SYSTEM TestMixerMain
  (* Version 1.0, 2024-03-03, ADMIN *)
  APPLICATION TestMixerMainApp
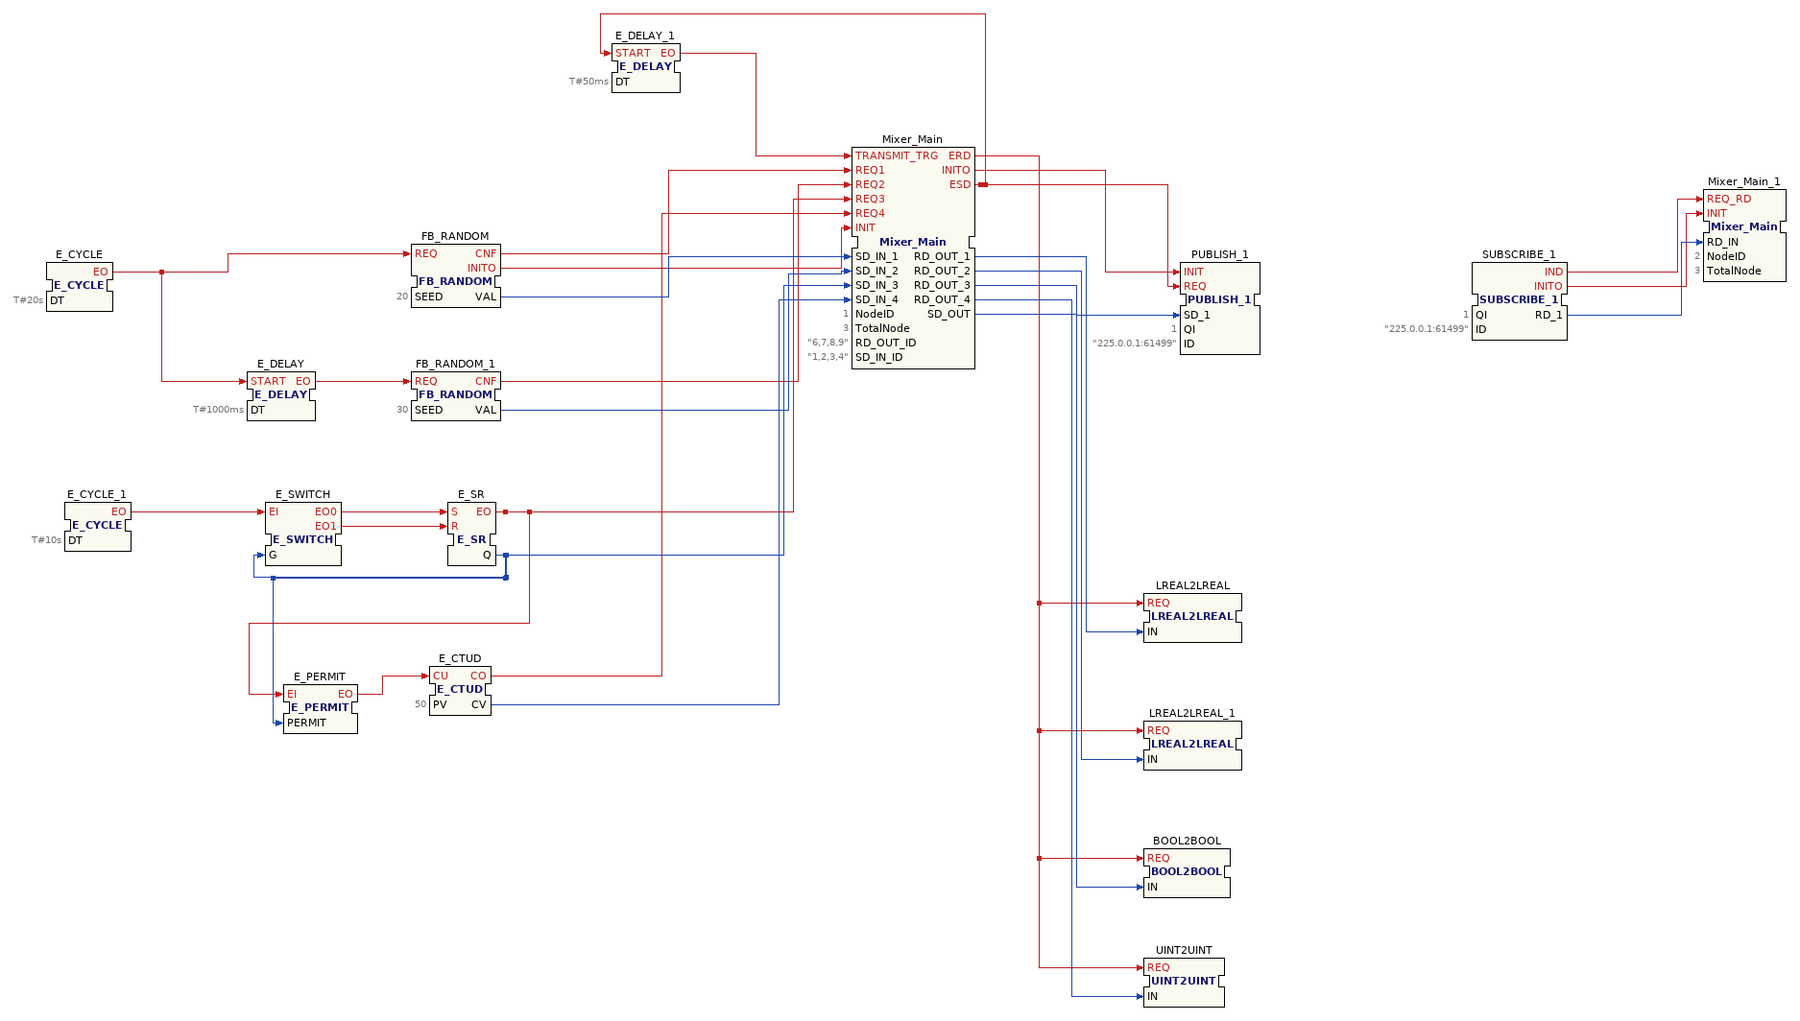
    FBS
      Mixer_Main : Mixer_Main(NodeID := 1, TotalNode := 3, RD_OUT_ID := "6,7,8,9", SD_IN_ID := "1,2,3,4");
      Mixer_Main_1 : Mixer_Main(NodeID := 2, TotalNode := 3);
      SUBSCRIBE_1 : SUBSCRIBE_1(QI := 1, ID := "225.0.0.1:61499");
      PUBLISH_1 : PUBLISH_1(QI := 1, ID := "225.0.0.1:61499");
      UINT2UINT : UINT2UINT;
      BOOL2BOOL : BOOL2BOOL;
      LREAL2LREAL_1 : LREAL2LREAL;
      LREAL2LREAL : LREAL2LREAL;
      E_DELAY_1 : E_DELAY(DT := T#50ms);
      E_CTUD : E_CTUD(PV := 50);
      E_PERMIT : E_PERMIT;
      FB_RANDOM : FB_RANDOM(SEED := 20);
      E_CYCLE_1 : E_CYCLE(DT := T#10s);
      E_SR : E_SR;
      E_SWITCH : E_SWITCH;
      FB_RANDOM_1 : FB_RANDOM(SEED := 30);
      E_DELAY : E_DELAY(DT := T#1000ms);
      E_CYCLE : E_CYCLE(DT := T#20s);
    END_FBS
    EVENT_CONNECTIONS
      Mixer_Main.ERD TO LREAL2LREAL.REQ;
      Mixer_Main.ERD TO LREAL2LREAL_1.REQ;
      Mixer_Main.ERD TO BOOL2BOOL.REQ;
      Mixer_Main.ERD TO UINT2UINT.REQ;
      Mixer_Main.INITO TO PUBLISH_1.INIT;
      Mixer_Main.ESD TO PUBLISH_1.REQ;
      Mixer_Main.ESD TO E_DELAY_1.START;
      E_DELAY_1.EO TO Mixer_Main.TRANSMIT_TRG;
      E_SWITCH.EO0 TO E_SR.S;
      E_CYCLE.EO TO E_DELAY.START;
      E_SWITCH.EO1 TO E_SR.R;
      E_CYCLE_1.EO TO E_SWITCH.EI;
      E_DELAY.EO TO FB_RANDOM_1.REQ;
      E_SR.EO TO E_PERMIT.EI;
      E_PERMIT.EO TO E_CTUD.CU;
      E_CYCLE.EO TO FB_RANDOM.REQ;
      FB_RANDOM.CNF TO Mixer_Main.REQ1;
      FB_RANDOM_1.CNF TO Mixer_Main.REQ2;
      E_SR.EO TO Mixer_Main.REQ3;
      E_CTUD.CO TO Mixer_Main.REQ4;
      SUBSCRIBE_1.IND TO Mixer_Main_1.REQ_RD;
      SUBSCRIBE_1.INITO TO Mixer_Main_1.INIT;
      FB_RANDOM.INITO TO Mixer_Main.INIT;
    END_CONNECTIONS
    DATA_CONNECTIONS
      Mixer_Main.RD_OUT_1 TO LREAL2LREAL.IN;
      Mixer_Main.RD_OUT_2 TO LREAL2LREAL_1.IN;
      Mixer_Main.RD_OUT_3 TO BOOL2BOOL.IN;
      Mixer_Main.RD_OUT_4 TO UINT2UINT.IN;
      Mixer_Main.SD_OUT TO PUBLISH_1.SD_1;
      E_SR.Q TO E_PERMIT.PERMIT;
      E_SR.Q TO E_SWITCH.G;
      FB_RANDOM.VAL TO Mixer_Main.SD_IN_1;
      FB_RANDOM_1.VAL TO Mixer_Main.SD_IN_2;
      E_SR.Q TO Mixer_Main.SD_IN_3;
      E_CTUD.CV TO Mixer_Main.SD_IN_4;
      SUBSCRIBE_1.RD_1 TO Mixer_Main_1.RD_IN;
    END_CONNECTIONS
  END_APPLICATION
  DEVICE FORTE_PC : FORTE_PC(MGR_ID := "localhost:61500")
    {SET_ATTRIBUTE(Profile, HOLOBLOC)} (* device profile *)
    RESOURCE EMB_RES : EMB_RES
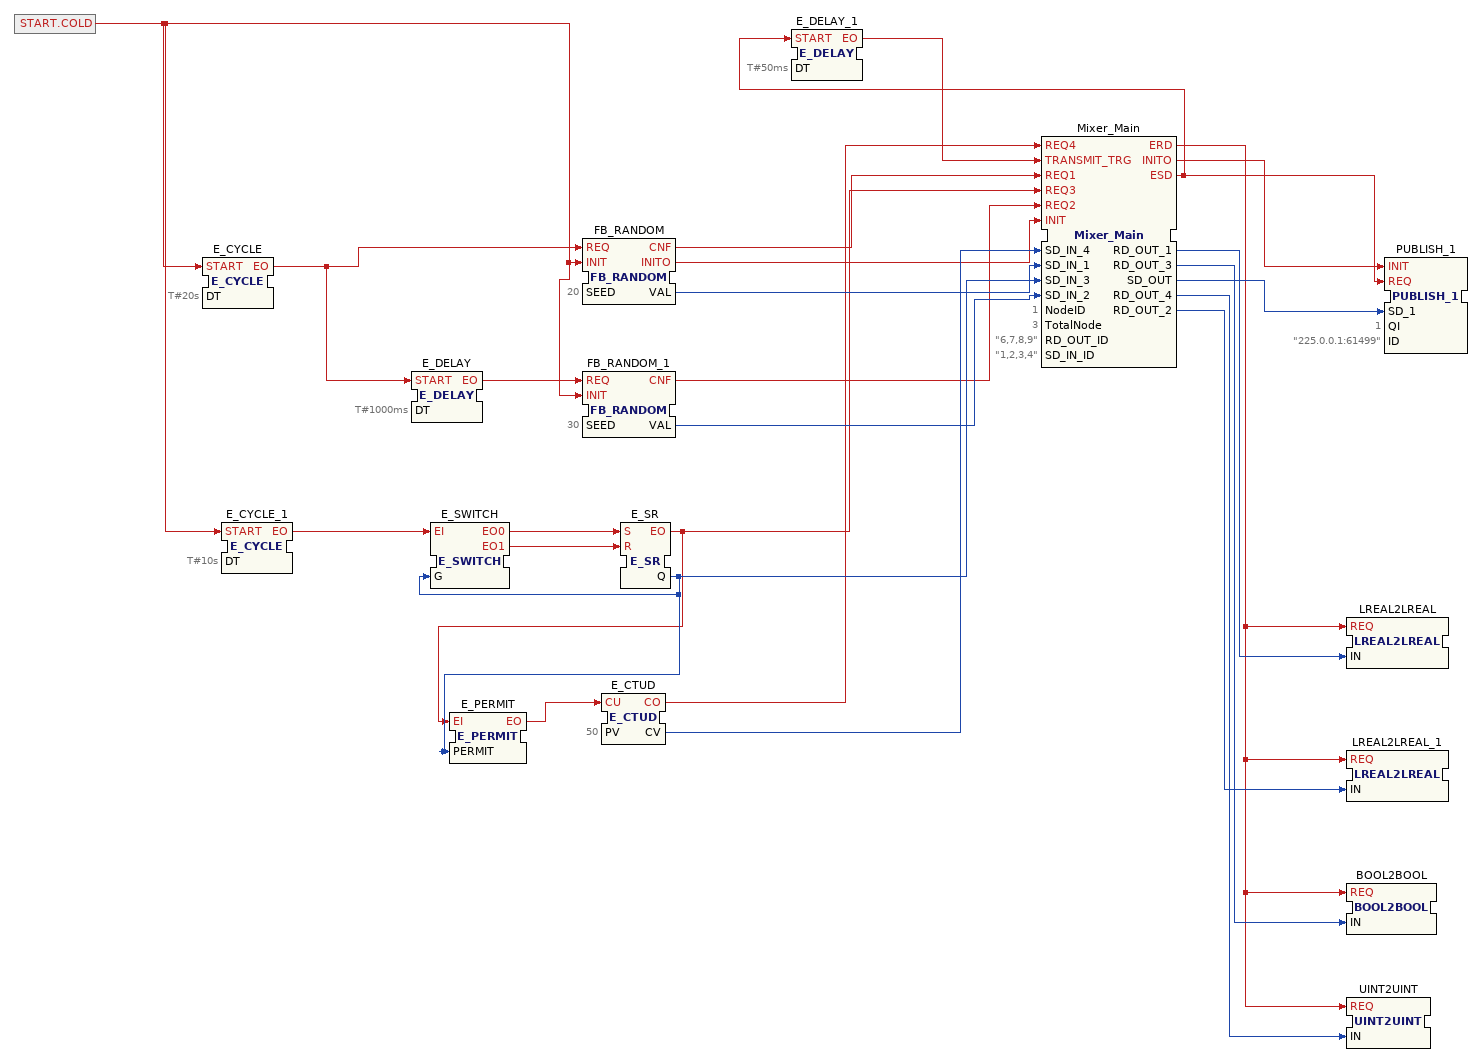
      FBS
        Mixer_Main : Mixer_Main(NodeID := 1, TotalNode := 3, RD_OUT_ID := "6,7,8,9", SD_IN_ID := "1,2,3,4");
        E_SWITCH : E_SWITCH;
        E_PERMIT : E_PERMIT;
        LREAL2LREAL : LREAL2LREAL;
        E_CTUD : E_CTUD(PV := 50);
        BOOL2BOOL : BOOL2BOOL;
        PUBLISH_1 : PUBLISH_1(QI := 1, ID := "225.0.0.1:61499");
        E_DELAY_1 : E_DELAY(DT := T#50ms);
        UINT2UINT : UINT2UINT;
        E_CYCLE : E_CYCLE(DT := T#20s);
        E_CYCLE_1 : E_CYCLE(DT := T#10s);
        FB_RANDOM : FB_RANDOM(SEED := 20);
        E_SR : E_SR;
        LREAL2LREAL_1 : LREAL2LREAL;
        FB_RANDOM_1 : FB_RANDOM(SEED := 30);
        E_DELAY : E_DELAY(DT := T#1000ms);
      END_FBS
      EVENT_CONNECTIONS
        Mixer_Main.ERD TO LREAL2LREAL.REQ;
        E_PERMIT.EO TO E_CTUD.CU;
        E_CTUD.CO TO Mixer_Main.REQ4;
        Mixer_Main.ERD TO BOOL2BOOL.REQ;
        Mixer_Main.INITO TO PUBLISH_1.INIT;
        Mixer_Main.ESD TO PUBLISH_1.REQ;
        Mixer_Main.ESD TO E_DELAY_1.START;
        E_DELAY_1.EO TO Mixer_Main.TRANSMIT_TRG;
        Mixer_Main.ERD TO UINT2UINT.REQ;
        E_CYCLE_1.EO TO E_SWITCH.EI;
        E_CYCLE.EO TO FB_RANDOM.REQ;
        FB_RANDOM.CNF TO Mixer_Main.REQ1;
        E_SWITCH.EO0 TO E_SR.S;
        E_SWITCH.EO1 TO E_SR.R;
        E_SR.EO TO E_PERMIT.EI;
        E_SR.EO TO Mixer_Main.REQ3;
        Mixer_Main.ERD TO LREAL2LREAL_1.REQ;
        FB_RANDOM_1.CNF TO Mixer_Main.REQ2;
        E_CYCLE.EO TO E_DELAY.START;
        E_DELAY.EO TO FB_RANDOM_1.REQ;
        START.COLD TO E_CYCLE.START;
        START.COLD TO FB_RANDOM.INIT;
        START.COLD TO FB_RANDOM_1.INIT;
        START.COLD TO E_CYCLE_1.START;
        FB_RANDOM.INITO TO Mixer_Main.INIT;
      END_CONNECTIONS
      DATA_CONNECTIONS
        Mixer_Main.RD_OUT_1 TO LREAL2LREAL.IN;
        E_CTUD.CV TO Mixer_Main.SD_IN_4;
        Mixer_Main.RD_OUT_3 TO BOOL2BOOL.IN;
        Mixer_Main.SD_OUT TO PUBLISH_1.SD_1;
        Mixer_Main.RD_OUT_4 TO UINT2UINT.IN;
        FB_RANDOM.VAL TO Mixer_Main.SD_IN_1;
        E_SR.Q TO E_PERMIT.PERMIT;
        E_SR.Q TO E_SWITCH.G;
        E_SR.Q TO Mixer_Main.SD_IN_3;
        Mixer_Main.RD_OUT_2 TO LREAL2LREAL_1.IN;
        FB_RANDOM_1.VAL TO Mixer_Main.SD_IN_2;
      END_CONNECTIONS
    END_RESOURCE
  END_DEVICE
  DEVICE FORTE_PC_1 : FORTE_PC(MGR_ID := "localhost:61501")
    {SET_ATTRIBUTE(Profile, HOLOBLOC)} (* device profile *)
    RESOURCE EMB_RES : EMB_RES
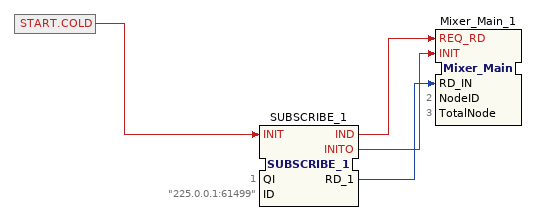
      FBS
        SUBSCRIBE_1 : SUBSCRIBE_1(QI := 1, ID := "225.0.0.1:61499");
        Mixer_Main_1 : Mixer_Main(NodeID := 2, TotalNode := 3);
      END_FBS
      EVENT_CONNECTIONS
        SUBSCRIBE_1.IND TO Mixer_Main_1.REQ_RD;
        SUBSCRIBE_1.INITO TO Mixer_Main_1.INIT;
        START.COLD TO SUBSCRIBE_1.INIT;
      END_CONNECTIONS
      DATA_CONNECTIONS
        SUBSCRIBE_1.RD_1 TO Mixer_Main_1.RD_IN;
      END_CONNECTIONS
    END_RESOURCE
  END_DEVICE
  MAPPINGS
    TestMixerMainApp.Mixer_Main ON FORTE_PC.EMB_RES.Mixer_Main;
    TestMixerMainApp.E_SWITCH ON FORTE_PC.EMB_RES.E_SWITCH;
    TestMixerMainApp.E_PERMIT ON FORTE_PC.EMB_RES.E_PERMIT;
    TestMixerMainApp.LREAL2LREAL ON FORTE_PC.EMB_RES.LREAL2LREAL;
    TestMixerMainApp.E_CTUD ON FORTE_PC.EMB_RES.E_CTUD;
    TestMixerMainApp.BOOL2BOOL ON FORTE_PC.EMB_RES.BOOL2BOOL;
    TestMixerMainApp.PUBLISH_1 ON FORTE_PC.EMB_RES.PUBLISH_1;
    TestMixerMainApp.E_DELAY_1 ON FORTE_PC.EMB_RES.E_DELAY_1;
    TestMixerMainApp.UINT2UINT ON FORTE_PC.EMB_RES.UINT2UINT;
    TestMixerMainApp.E_CYCLE ON FORTE_PC.EMB_RES.E_CYCLE;
    TestMixerMainApp.E_CYCLE_1 ON FORTE_PC.EMB_RES.E_CYCLE_1;
    TestMixerMainApp.FB_RANDOM ON FORTE_PC.EMB_RES.FB_RANDOM;
    TestMixerMainApp.E_SR ON FORTE_PC.EMB_RES.E_SR;
    TestMixerMainApp.LREAL2LREAL_1 ON FORTE_PC.EMB_RES.LREAL2LREAL_1;
    TestMixerMainApp.FB_RANDOM_1 ON FORTE_PC.EMB_RES.FB_RANDOM_1;
    TestMixerMainApp.E_DELAY ON FORTE_PC.EMB_RES.E_DELAY;
    TestMixerMainApp.SUBSCRIBE_1 ON FORTE_PC_1.EMB_RES.SUBSCRIBE_1;
    TestMixerMainApp.Mixer_Main_1 ON FORTE_PC_1.EMB_RES.Mixer_Main_1;
  END_MAPPINGS
  SEGMENTS
    Ethernet : Ethernet;
  END_SEGMENTS
  LINKS
    FORTE_PC => Ethernet;
    FORTE_PC_1 => Ethernet;
  END_LINKS
END_SYSTEM
